INTERFACE I_Object

METHOD RegisterWithParent
VAR_INPUT
	Runner : I_HostObjects;
END_VAR
END_METHOD

END_INTERFACE

(* stored: Version 1.1.0.1
   Itf I_Object: Id {cc5f09b5-b4c7-477b-9761-d6fd857f7e64}
   Method RegisterWithParent: Id {a872b065-77ae-4022-8c54-eeadc17c5447} *)
